// Mitsubishi GX Works2 project: connect   PLC: Q03UDV

PROGRAM MAIN
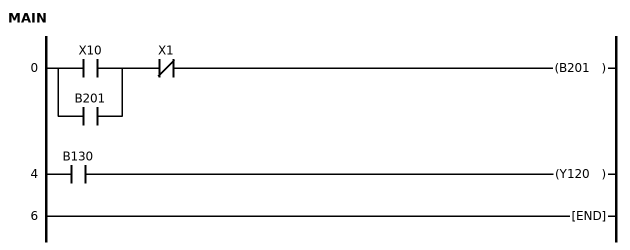
0     LD      X10
      OR      B201
      ANI     X1
      OUT     B201
4     LD      B130
      OUT     Y120
6     END
END_PROGRAM
